// TIA Portal V17 export
// export: Created 2023-02-25T16:31:53.3277457Z, ExportSetting WithDefaults, DisplayName Totally Integrated Automation Portal, DisplayVersion V17, DisplayName TIA Portal Openness, DisplayVersion V17, DisplayName TIA Portal Version Control Interface, DisplayVersion V17, DisplayName TIA Portal Test Suite Advanced, DisplayVersion V17, DisplayName STEP 7 Professional, DisplayVersion V17, DisplayName SIMATIC Energy Suite, DisplayVersion V17, DisplayName STEP 7 Safety, DisplayVersion V17, DisplayName WinCC Professional, DisplayVersion V17
FUNCTION "LOG_ColumnLight" : Void   // FC16, LAD
{ S7_Optimized_Access := 'TRUE' }
VERSION : 0.1
// stored: AutoNumber true, IsIECCheckEnabled false, SetENOAutomatically false, UDAEnableTagReadback false
   VAR_TEMP
      Green_1 : Bool;
      Green_2 : Bool;
      Yellow_1 : Bool;
      Yellow_2 : Bool;
   END_VAR
BEGIN

REGION Network 1: Start line manual mode signaling
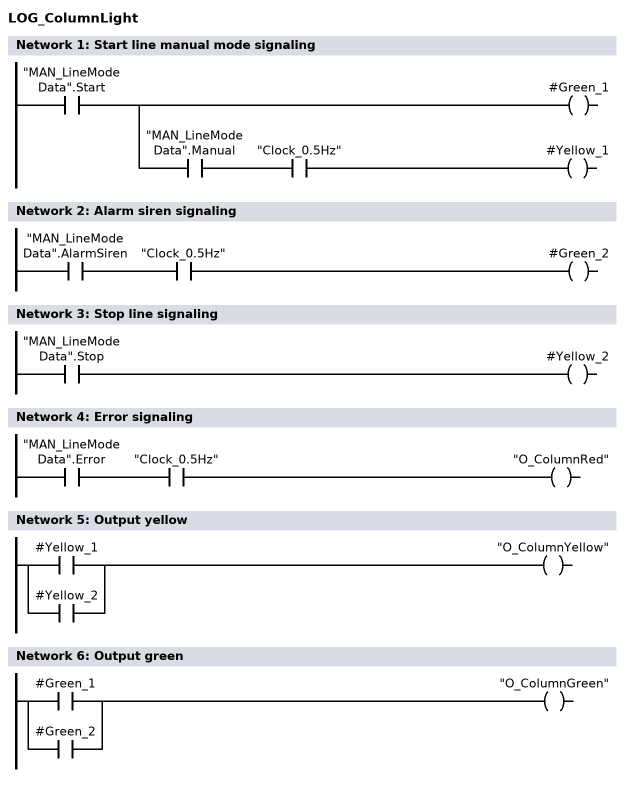
   RUNG wire#powerrail
      Contact( "MAN_LineModeData".Start )
      wire#w1
      Coil( #Green_1 )
   END_RUNG
   RUNG wire#w1
      Contact( "MAN_LineModeData".Manual )
      Contact( "Clock_0.5Hz" )
      Coil( #Yellow_1 )
   END_RUNG
   // the same network as SCL:
   #Green_1 := "MAN_LineModeData".Start;
   #Yellow_1 := "MAN_LineModeData".Start AND "MAN_LineModeData".Manual AND "Clock_0.5Hz";
END_REGION

REGION Network 2: Alarm siren signaling
   RUNG wire#powerrail
      Contact( "MAN_LineModeData".AlarmSiren )
      Contact( "Clock_0.5Hz" )
      Coil( #Green_2 )
   END_RUNG
   // the same network as SCL:
   #Green_2 := "MAN_LineModeData".AlarmSiren AND "Clock_0.5Hz";
END_REGION

REGION Network 3: Stop line signaling
   RUNG wire#powerrail
      Contact( "MAN_LineModeData".Stop )
      Coil( #Yellow_2 )
   END_RUNG
   // the same network as SCL:
   #Yellow_2 := "MAN_LineModeData".Stop;
END_REGION

REGION Network 4: Error signaling
   RUNG wire#powerrail
      Contact( "MAN_LineModeData".Error )
      Contact( "Clock_0.5Hz" )
      Coil( "O_ColumnRed" )
   END_RUNG
   // the same network as SCL:
   "O_ColumnRed" := "MAN_LineModeData".Error AND "Clock_0.5Hz";
END_REGION

REGION Network 5: Output yellow
   RUNG wire#powerrail
      Contact( #Yellow_1 )
      wire#w1
      Coil( "O_ColumnYellow" )
   END_RUNG
   RUNG wire#powerrail
      Contact( #Yellow_2 )
   END_RUNG wire#w1
   // the same network as SCL:
   "O_ColumnYellow" := #Yellow_1 OR #Yellow_2;
END_REGION

REGION Network 6: Output green
   RUNG wire#powerrail
      Contact( #Green_1 )
      wire#w1
      Coil( "O_ColumnGreen" )
   END_RUNG
   RUNG wire#powerrail
      Contact( #Green_2 )
   END_RUNG wire#w1
   // the same network as SCL:
   "O_ColumnGreen" := #Green_1 OR #Green_2;
END_REGION
END_FUNCTION
